FUNCTION_BLOCK HASH (* Basic Function Block Type *)
  (* Standard: 61499-2 *)
  (* Version 0.0, 4/22/2025, SESA66148, Template *)
  PACKAGE SEFR.HashTools;
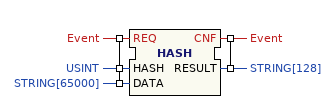
  EVENT_INPUT
    REQ WITH HASH, DATA; (* Normal Execution Request *)
  END_EVENT
  EVENT_OUTPUT
    CNF WITH RESULT; (* Execution Confirmation *)
  END_EVENT
  VAR_INPUT
    HASH : USINT; (* 0=MD5 | 1=SHA1 | 2=SHA224 | 3=SHA256 | 4=SHA384 | 5=SHA512 | 6=SHA512_224 | 7=SHA512_256 *) {SET_ATTRIBUTE(ParameterEditor, ComboBox{Enums=MD5 = 0|SHA1 = 1|SHA224 = 2|SHA256 = 3|SHA384 = 4|SHA512 = 5|SHA512_224 = 6|SHA512_256 = 7$})}
    DATA : STRING[65000];
  END_VAR
  VAR_OUTPUT
    RESULT : STRING[128];
  END_VAR
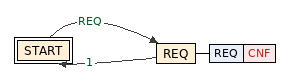
  EC_STATES
    START; (* Initial State *)
    REQ : REQ -> CNF; (* Normal execution *)
  END_STATES
  EC_TRANSITIONS
    START TO REQ := REQ;
    REQ TO START := 1;
  END_TRANSITIONS
  ALGORITHM REQ IN ST: (* Normally executed algorithm *)
CASE HASH OF
	0: RESULT := HASH_MD5(DATA);
	1: RESULT := HASH_SHA1(DATA);
	2: RESULT := HASH_SHA224(DATA);
	3: RESULT := HASH_SHA256(DATA);
	4: RESULT := HASH_SHA384(DATA);
	5: RESULT := HASH_SHA512(DATA);
	6: RESULT := HASH_SHA512_224(DATA);
	7: RESULT := HASH_SHA512_256(DATA);
ELSE
	RESULT := '';
END_CASE;
  END_ALGORITHM
END_FUNCTION_BLOCK
